FUNCTION_BLOCK _STRING_TestSuite EXTENDS TcUnit.FB_TestSuite
VAR
END_VAR

TestAddress();
TestClearReference();
TestClone();
TestTypeNameReturnsExpected();
TestMakeReferenceToFollowsReference();
TestMakeReferenceToUpdatesReference();
TestSize();
TestValueReturnsExpectedAfterInit();
TestValueReturnsExpectedAfterChange();
TestSerializeTypeWith();
TestSerializeWith();
TestTryDeserializeFrom();
TestTryMakeReferenceToFollowsReference();
TestTryMakeReferenceToUpdatesReference();

METHOD PUBLIC TestAddress
VAR
    _type : _STRING('');
    notExpected : PVOID := 0;
    actual : PVOID;
END_VAR
TEST('TestAddress');

actual := _type.Address;

AssertFalse(
    Condition := (notExpected = actual),
    Message := 'Type did not return a valid address.'
);

TEST_FINISHED();
END_METHOD

METHOD PUBLIC TestClearReference
VAR
    _type : _STRING('');
	target : T_MaxString := '';
    expected : T_MaxString := '';
    actual : T_MaxString;
END_VAR
TEST('TestClearReference');

_type.MakeReferenceTo(target);
_type.ClearReference();
target := '123';

actual := _type.Value;

AssertEquals_STRING(
    Expected := expected,
    Actual := actual,
    Message := 'Value incorrectly followed target change'
);

TEST_FINISHED();
END_METHOD

METHOD PUBLIC TestClone
VAR
    _type : _STRING('123');
	clone : I_Datatype;
	isValidClone : BOOL;
	compareResult : DINT;
END_VAR
TEST('TestClone');

clone := _type.Clone();

isValidClone := clone <> 0;

IF isValidClone THEN
	compareResult := memcmp(_type.Address, clone.Address, clone.Size);
END_IF

AssertTrue(
	Condition := isValidClone,
	Message := 'Clone did not produce a clone'
);

AssertEquals_DINT(
	Expected := 0,
    Actual := compareResult,
    Message := 'Clone did not return a valid clone.'
);

clone.Dispose();

TEST_FINISHED();
END_METHOD

METHOD PUBLIC TestMakeReferenceToFollowsReference
VAR
    _type : _STRING('');
	target : T_MaxString := '';
    expected : T_MaxString := '123';
    actual : T_MaxString;
END_VAR
TEST('TestMakeReferenceToFollowsReference');

_type.MakeReferenceTo(target);
target := '123';

actual := _type.Value;

AssertEquals_STRING(
    Expected := expected,
    Actual := actual,
    Message := 'Value did not follow target change'
);

TEST_FINISHED();
END_METHOD

METHOD PUBLIC TestMakeReferenceToUpdatesReference
VAR
    _type : _STRING('');
	target : T_MaxString := '';
    expected : T_MaxString := '123';
    actual : T_MaxString;
END_VAR
TEST('TestMakeReferenceToUpdatesReference');

_type.MakeReferenceTo(target);
_type.Value := '123';

actual := target;

AssertEquals_STRING(
    Expected := expected,
    Actual := actual,
    Message := 'Value did not update target'
);

TEST_FINISHED();
END_METHOD

METHOD PUBLIC TestSerializeTypeWith
VAR
    _type : _STRING('');
    serializer : JsonSerializer;
    expected : STRING := '{"typeName":"STRING"}';
    actual : STRING(500);
END_VAR
TEST('TestSerializeTypeWith');

serializer.Reset();
_type.SerializeTypeWith(serializer);
serializer.TryGetSerializedData(ADR(actual), SIZEOF(actual));

AssertEquals_STRING(
    Expected := expected,
    Actual := actual,
    Message := 'Serialization of type did not return correct string.'
);

TEST_FINISHED();
END_METHOD

METHOD PUBLIC TestSerializeWith
VAR
    _type : _STRING('abcdefghijklmnopqrstuvwxyzABCDEFGHIJKLMNOPQRSTUVWXYZ01234567890');
    serializer : JsonSerializer;
    expected : STRING := '"abcdefghijklmnopqrstuvwxyzABCDEFGHIJKLMNOPQRSTUVWXYZ01234567890"';
    actual : STRING(500);
END_VAR
TEST('TestSerializeWith');

serializer.Reset();
_type.SerializeWith(serializer);
serializer.TryGetSerializedData(ADR(actual), SIZEOF(actual));

AssertEquals_STRING(
    Expected := expected,
    Actual := actual,
    Message := 'Serialization of type data did not return correct string.'
);

TEST_FINISHED();
END_METHOD

METHOD PUBLIC TestSize
VAR
    _type : _STRING('');
    expected : UDINT := SIZEOF(T_MaxString);
    actual : UDINT;
END_VAR
TEST('TestSize');

actual := _type.Size;

AssertEquals_UDINT(
    Expected := Expected,
    Actual := actual,
    Message := 'Type did not return the correct size.'
);

TEST_FINISHED();
END_METHOD

METHOD PUBLIC TestTryDeserializeFrom
VAR
    deserializer : JsonDeserializer;
    feedback : DeserializerFeedback;
    json : STRING := '"abcdefghijklmnopqrstuvwxyzABCDEFGHIJKLMNOPQRSTUVWXYZ01234567890"';
    _type : _STRING('');
    expected : T_MaxString := 'abcdefghijklmnopqrstuvwxyzABCDEFGHIJKLMNOPQRSTUVWXYZ01234567890';
    actual : T_MaxString;
 END_VAR
TEST('TestTryDeserializeFrom');

deserializer.Reset();
deserializer.TryLoad(json);
_type.TryDeserializeFrom(Deserializer, Feedback);

actual := _type.Value;

AssertEquals_STRING(
    Expected := expected,
    Actual := actual,
    Message := 'Type did not deserialize correctly.'
);

TEST_FINISHED();
END_METHOD

METHOD PUBLIC TestTryMakeReferenceToFollowsReference
VAR
    _type : _STRING('');
	target : _STRING('');
    expected : T_MaxString := '123';
    actual : T_MaxString;
END_VAR
TEST('TestTryMakeReferenceToFollowsReference');

_type.TryMakeReferenceTo(target);
target.Value := '123';

actual := _type.Value;

AssertEquals_STRING(
    Expected := expected,
    Actual := actual,
    Message := 'Value did not follow target change'
);

TEST_FINISHED();
END_METHOD

METHOD PUBLIC TestTryMakeReferenceToUpdatesReference
VAR
    _type : _STRING('');
	target : _STRING('');
    expected : T_MaxString := '123';
    actual : T_MaxString;
END_VAR
TEST('TestTryMakeReferenceToUpdatesReference');

_type.TryMakeReferenceTo(target);
_type.Value := '123';

actual := target.Value;

AssertEquals_STRING(
    Expected := expected,
    Actual := actual,
    Message := 'Value did not update target'
);

TEST_FINISHED();
END_METHOD

METHOD PUBLIC TestTypeNameReturnsExpected
VAR
    _type : _STRING('');
    expected : STRING := 'STRING';
    actual : STRING;
END_VAR
TEST('TestTypeNameReturnsExpected');

actual := _type.TypeName;

AssertEquals_STRING(
    Expected := expected,
    Actual := actual,
    Message := 'Type did not return correct iec type.'
);

TEST_FINISHED();
END_METHOD

METHOD PUBLIC TestValueReturnsExpectedAfterChange
VAR
    _type : _STRING('');
    expected : T_MaxString := '123';
    actual : T_MaxString;
END_VAR
TEST('TestValueReturnsExpectedAfterChange');

_type.Value := '123';

actual := _type.Value;

AssertEquals_STRING(
    Expected := expected,
    Actual := actual,
    Message := 'Expected value not returned after change.'
);

TEST_FINISHED();
END_METHOD

METHOD PUBLIC TestValueReturnsExpectedAfterInit
VAR
    _type : _STRING('123');
    expected : T_MaxString := '123';
    actual : T_MaxString;
END_VAR
TEST('TestValueReturnsExpectedAfterInit');

actual := _type.Value;

AssertEquals_STRING(
    Expected := expected,
    Actual := actual,
    Message := 'Expected value not returned after Init.'
);

TEST_FINISHED();
END_METHOD

END_FUNCTION_BLOCK

(* stored: Version 1.1.0.1, ProductVersion 3.1.4024.12
   POU _STRING_TestSuite: Id {bdaf3f65-5b06-0a15-1b8a-4308e354a882}, SpecialFunc None
   Method TestAddress: Id {2b9e3bfe-2fe8-0566-34af-aa05646b5639}
   Method TestClearReference: Id {ac032fe2-fccb-0a17-231e-0633546ca80e}
   Method TestClone: Id {5bcdeab5-a5a6-09b8-2946-62ba6a741281}
   Method TestMakeReferenceToFollowsReference: Id {b7ac241b-aa18-01f2-3433-42794682e7a2}
   Method TestMakeReferenceToUpdatesReference: Id {7a6a6c64-287d-0f90-1dce-60d85acd9b27}
   Method TestSerializeTypeWith: Id {d8af1417-bd7e-039f-014c-c4e88dbff48e}
   Method TestSerializeWith: Id {02733de1-d55f-0cd8-3486-d792465b53ee}
   Method TestSize: Id {76cd5de1-ed54-0f1f-29ee-4871080eec77}
   Method TestTryDeserializeFrom: Id {0f39ff36-c5a1-0558-113b-2df682bae70b}
   Method TestTryMakeReferenceToFollowsReference: Id {d63d3abf-940e-0da3-079a-aa79c1190211}
   Method TestTryMakeReferenceToUpdatesReference: Id {db00c639-116f-044f-384d-67b60756ee18}
   Method TestTypeNameReturnsExpected: Id {c1ff6c08-f76b-072d-287b-c4a51cb5dfdd}
   Method TestValueReturnsExpectedAfterChange: Id {f61aaa6d-78a2-06b6-3141-0413889047fb}
   Method TestValueReturnsExpectedAfterInit: Id {9e4c65a2-fc11-00f6-1a98-5c0a753e628b} *)
